PROGRAM P_ADS_Gauge
VAR
	bTrigger				: BOOL;
	lr_weight_1				:LREAL;
	lr_weight_2				:LREAL;
	lr_weight_3				:LREAL;
	lr_weight_4				:LREAL;
	
	lr_correction_weight_1  :LREAL;
	lr_correction_weight_2  :LREAL;
	lr_correction_weight_3  :LREAL;
	lr_correction_weight_4  :LREAL;	
	
	lr_dosed_1				:LREAL;
	lr_dosed_2				:LREAL;
	lr_dosed_3				:LREAL;
	lr_dosed_4				:LREAL;
	
	isensor_value_1			:INT;
	isensor_value_2			:INT;
	
	lr_screwer_torque_1		:LREAL;
	lr_screwer_torque_2		:LREAL;
	lr_screwer_torque_set	:LREAL;
	lr_screwer_torque_set_2	:LREAL;
//weight measureg
	fbRead_1: FB_ReadAdsSymByName;
	fbRead_2: FB_ReadAdsSymByName;
	fbRead_3: FB_ReadAdsSymByName;
	fbRead_4: FB_ReadAdsSymByName;
//correction weight	
	fbRead_5: FB_ReadAdsSymByName;
	fbRead_6: FB_ReadAdsSymByName;
	fbRead_7: FB_ReadAdsSymByName;
	fbRead_8: FB_ReadAdsSymByName;
//dose volume
	fbRead_9: FB_ReadAdsSymByName;
	fbRead_10: FB_ReadAdsSymByName;
	fbRead_11: FB_ReadAdsSymByName;
	fbRead_12: FB_ReadAdsSymByName;
//tank level
	fbRead_13: FB_ReadAdsSymByName;
	fbRead_14: FB_ReadAdsSymByName;
//Screwer torque
	fbRead_17: FB_ReadAdsSymByName;
	fbRead_16: FB_ReadAdsSymByName;
//Screwer torque recipe
	fbRead_15: FB_ReadAdsSymByName;
	fbRead_18: FB_ReadAdsSymByName;
	
	fbCyclicReadout: TON;
END_VAR

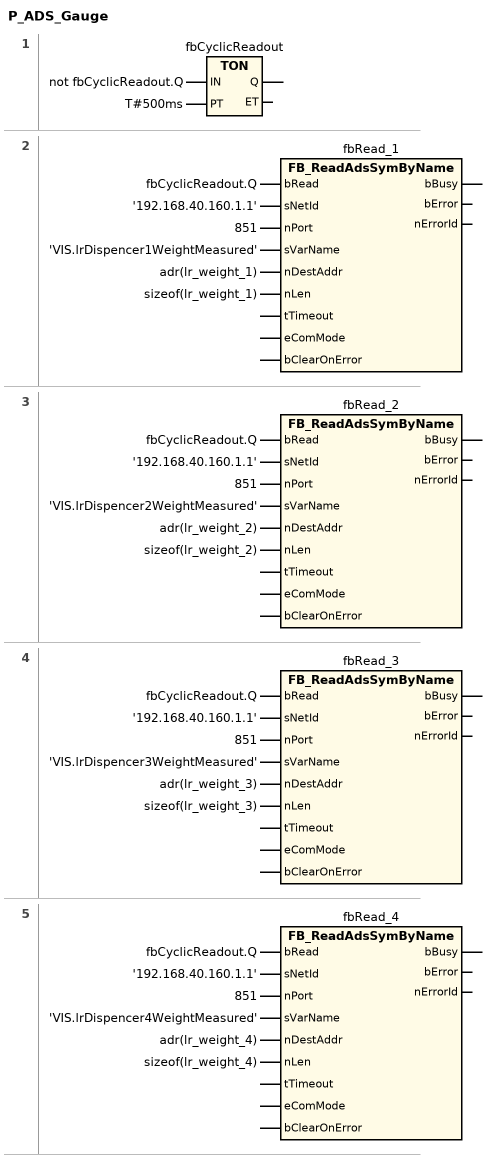
// NETWORK 1
fbCyclicReadout(IN := not fbCyclicReadout.Q, PT := T#500ms); // TON

// NETWORK 2
fbRead_1(
    bRead := fbCyclicReadout.Q,
    sNetId := '192.168.40.160.1.1',
    nPort := 851,
    sVarName := 'VIS.lrDispencer1WeightMeasured',
    nDestAddr := adr(lr_weight_1),
    nLen := sizeof(lr_weight_1)); // FB_ReadAdsSymByName

// NETWORK 3
fbRead_2(
    bRead := fbCyclicReadout.Q,
    sNetId := '192.168.40.160.1.1',
    nPort := 851,
    sVarName := 'VIS.lrDispencer2WeightMeasured',
    nDestAddr := adr(lr_weight_2),
    nLen := sizeof(lr_weight_2)); // FB_ReadAdsSymByName

// NETWORK 4
fbRead_3(
    bRead := fbCyclicReadout.Q,
    sNetId := '192.168.40.160.1.1',
    nPort := 851,
    sVarName := 'VIS.lrDispencer3WeightMeasured',
    nDestAddr := adr(lr_weight_3),
    nLen := sizeof(lr_weight_3)); // FB_ReadAdsSymByName

// NETWORK 5
fbRead_4(
    bRead := fbCyclicReadout.Q,
    sNetId := '192.168.40.160.1.1',
    nPort := 851,
    sVarName := 'VIS.lrDispencer4WeightMeasured',
    nDestAddr := adr(lr_weight_4),
    nLen := sizeof(lr_weight_4)); // FB_ReadAdsSymByName

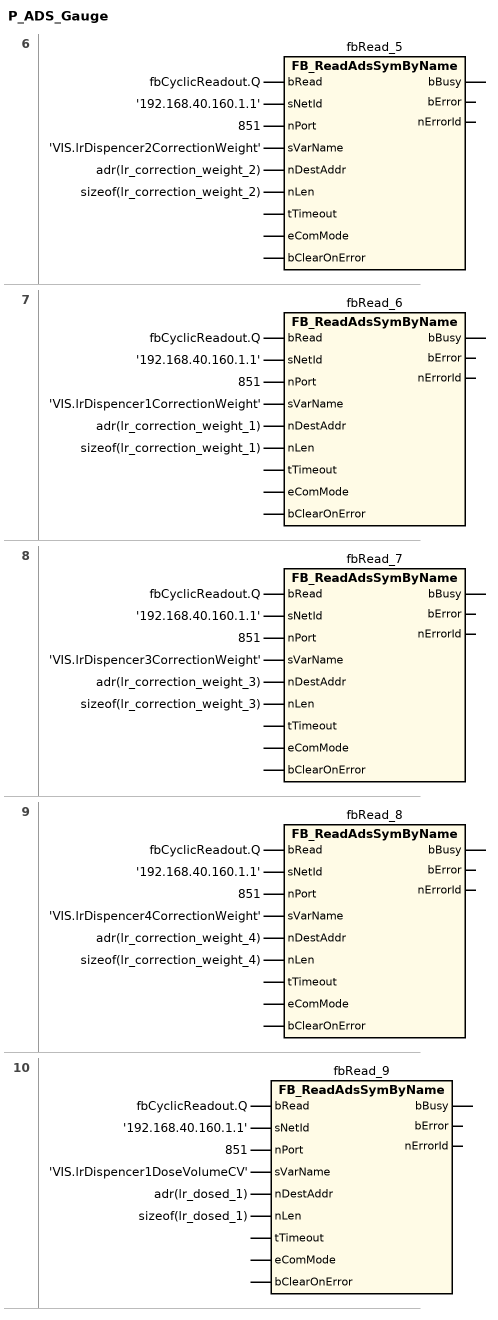
// NETWORK 6
fbRead_5(
    bRead := fbCyclicReadout.Q,
    sNetId := '192.168.40.160.1.1',
    nPort := 851,
    sVarName := 'VIS.lrDispencer2CorrectionWeight',
    nDestAddr := adr(lr_correction_weight_2),
    nLen := sizeof(lr_correction_weight_2)); // FB_ReadAdsSymByName

// NETWORK 7
fbRead_6(
    bRead := fbCyclicReadout.Q,
    sNetId := '192.168.40.160.1.1',
    nPort := 851,
    sVarName := 'VIS.lrDispencer1CorrectionWeight',
    nDestAddr := adr(lr_correction_weight_1),
    nLen := sizeof(lr_correction_weight_1)); // FB_ReadAdsSymByName

// NETWORK 8
fbRead_7(
    bRead := fbCyclicReadout.Q,
    sNetId := '192.168.40.160.1.1',
    nPort := 851,
    sVarName := 'VIS.lrDispencer3CorrectionWeight',
    nDestAddr := adr(lr_correction_weight_3),
    nLen := sizeof(lr_correction_weight_3)); // FB_ReadAdsSymByName

// NETWORK 9
fbRead_8(
    bRead := fbCyclicReadout.Q,
    sNetId := '192.168.40.160.1.1',
    nPort := 851,
    sVarName := 'VIS.lrDispencer4CorrectionWeight',
    nDestAddr := adr(lr_correction_weight_4),
    nLen := sizeof(lr_correction_weight_4)); // FB_ReadAdsSymByName

// NETWORK 10
fbRead_9(
    bRead := fbCyclicReadout.Q,
    sNetId := '192.168.40.160.1.1',
    nPort := 851,
    sVarName := 'VIS.lrDispencer1DoseVolumeCV',
    nDestAddr := adr(lr_dosed_1),
    nLen := sizeof(lr_dosed_1)); // FB_ReadAdsSymByName

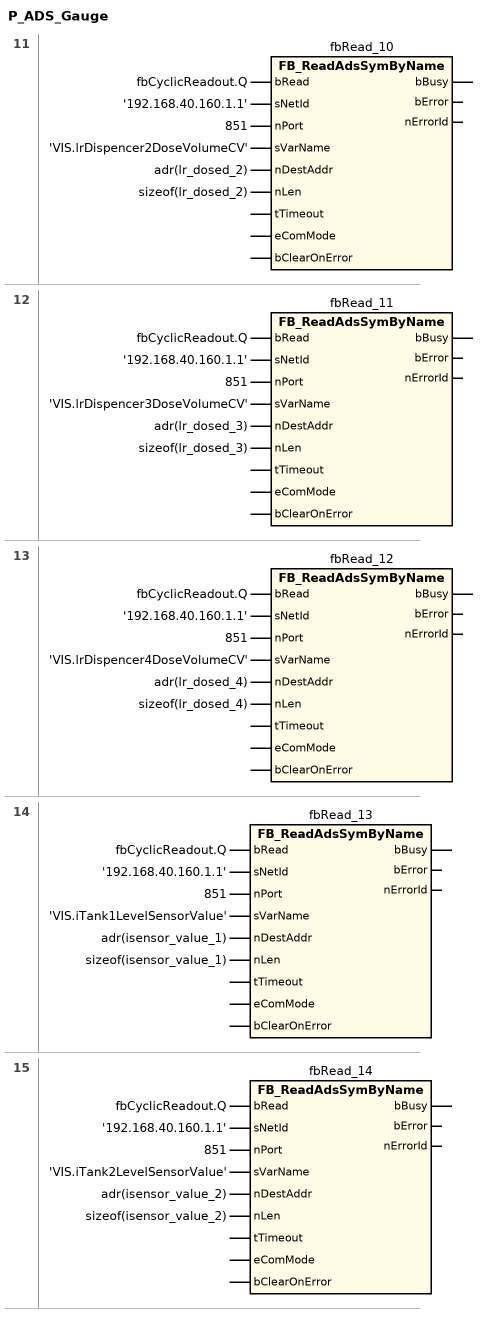
// NETWORK 11
fbRead_10(
    bRead := fbCyclicReadout.Q,
    sNetId := '192.168.40.160.1.1',
    nPort := 851,
    sVarName := 'VIS.lrDispencer2DoseVolumeCV',
    nDestAddr := adr(lr_dosed_2),
    nLen := sizeof(lr_dosed_2)); // FB_ReadAdsSymByName

// NETWORK 12
fbRead_11(
    bRead := fbCyclicReadout.Q,
    sNetId := '192.168.40.160.1.1',
    nPort := 851,
    sVarName := 'VIS.lrDispencer3DoseVolumeCV',
    nDestAddr := adr(lr_dosed_3),
    nLen := sizeof(lr_dosed_3)); // FB_ReadAdsSymByName

// NETWORK 13
fbRead_12(
    bRead := fbCyclicReadout.Q,
    sNetId := '192.168.40.160.1.1',
    nPort := 851,
    sVarName := 'VIS.lrDispencer4DoseVolumeCV',
    nDestAddr := adr(lr_dosed_4),
    nLen := sizeof(lr_dosed_4)); // FB_ReadAdsSymByName

// NETWORK 14
fbRead_13(
    bRead := fbCyclicReadout.Q,
    sNetId := '192.168.40.160.1.1',
    nPort := 851,
    sVarName := 'VIS.iTank1LevelSensorValue',
    nDestAddr := adr(isensor_value_1),
    nLen := sizeof(isensor_value_1)); // FB_ReadAdsSymByName

// NETWORK 15
fbRead_14(
    bRead := fbCyclicReadout.Q,
    sNetId := '192.168.40.160.1.1',
    nPort := 851,
    sVarName := 'VIS.iTank2LevelSensorValue',
    nDestAddr := adr(isensor_value_2),
    nLen := sizeof(isensor_value_2)); // FB_ReadAdsSymByName

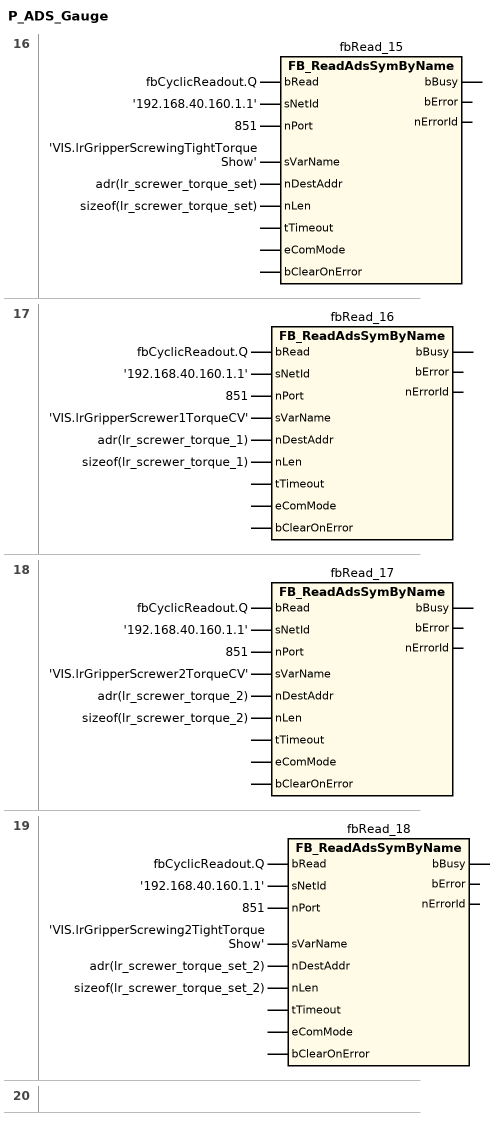
// NETWORK 16
fbRead_15(
    bRead := fbCyclicReadout.Q,
    sNetId := '192.168.40.160.1.1',
    nPort := 851,
    sVarName := 'VIS.lrGripperScrewingTightTorqueShow',
    nDestAddr := adr(lr_screwer_torque_set),
    nLen := sizeof(lr_screwer_torque_set)); // FB_ReadAdsSymByName

// NETWORK 17
fbRead_16(
    bRead := fbCyclicReadout.Q,
    sNetId := '192.168.40.160.1.1',
    nPort := 851,
    sVarName := 'VIS.lrGripperScrewer1TorqueCV',
    nDestAddr := adr(lr_screwer_torque_1),
    nLen := sizeof(lr_screwer_torque_1)); // FB_ReadAdsSymByName

// NETWORK 18
fbRead_17(
    bRead := fbCyclicReadout.Q,
    sNetId := '192.168.40.160.1.1',
    nPort := 851,
    sVarName := 'VIS.lrGripperScrewer2TorqueCV',
    nDestAddr := adr(lr_screwer_torque_2),
    nLen := sizeof(lr_screwer_torque_2)); // FB_ReadAdsSymByName

// NETWORK 19
fbRead_18(
    bRead := fbCyclicReadout.Q,
    sNetId := '192.168.40.160.1.1',
    nPort := 851,
    sVarName := 'VIS.lrGripperScrewing2TightTorqueShow',
    nDestAddr := adr(lr_screwer_torque_set_2),
    nLen := sizeof(lr_screwer_torque_set_2)); // FB_ReadAdsSymByName

// NETWORK 20

END_PROGRAM

(* stored: Version 1.1.0.1, ProductVersion 3.1.4024.12
   POU P_ADS_Gauge: Id {237a400d-a3ad-40e8-a01b-2c449190ee22}, SpecialFunc None *)
